Fanuc TP program (LS listing): GRIP_1_OPEN.LS

/PROG  GRIP_1_OPEN	  Macro
/ATTR
OWNER		= MNEDITOR;
COMMENT		= "Grip1Open";
PROG_SIZE	= 189;
CREATE		= DATE 19-12-09  TIME 17:51:00;
MODIFIED	= DATE 19-12-09  TIME 17:51:00;
FILE_NAME	= ;
VERSION		= 0;
LINE_COUNT	= 2;
MEMORY_SIZE	= 553;
PROTECT		= READ_WRITE;
TCD:  STACK_SIZE	= 0,
      TASK_PRIORITY	= 50,
      TIME_SLICE	= 0,
      BUSY_LAMP_OFF	= 0,
      ABORT_REQUEST	= 0,
      PAUSE_REQUEST	= 0;
DEFAULT_GROUP	= 1,*,*,*,*;
CONTROL_CODE	= 00000000 00000000;
/APPL
/APPL

AUTO_SINGULARITY_HEADER;
  ENABLE_SINGULARITY_AVOIDANCE   : TRUE;
/MN
   1:  RO[1:Open Gripper]=ON ;
   2:  WAIT R[15] ;
/POS
/END
